// TIA Portal V20 export
VAR_GLOBAL   // PLC tag table "PLC_Production_And_Rework"
   Emergency_Stop_Release AT %I0.0 : Bool;
   Sensor_Water_Fountain_Before_Entrace_Functional_Test_Spinner_Conveyor_Belt AT %I0.1 : Bool;
   Sensor_Water_Fountain_Entrace_Functional_Test_Spinner_Conveyor_Belt AT %I0.2 : Bool;
   Sensor_Water_Fountain_Entrace_Functional_Test_After_Spinner_Conveyor_Belt AT %I0.3 : Bool;
   Trigger_Read_Serial_Number_Entrace_Functional_Test AT %I0.4 : Bool;
   Sensor_Water_Fountain_Geting_Exit_Rework_Conveyor_Belt AT %I0.5 : Bool;
   Button_Water_Fountain_Get_Exit_Rework_Conveyor_Belt AT %I0.6 : Bool;
   Trigger_Read_Serial_Number_Exit_Functional_Test AT %I0.7 : Bool;
   Sensor_Water_Fountain_Exit_Functional_Test_Spinner_Conveyor_Belt AT %I1.0 : Bool;
   Sensor_Water_Fountain_Exit_Functional_Test_After_Spinner_Conveyor_Belt AT %I1.1 : Bool;
   Sensor_Water_Fountain_Geting_Entrace_Rework_Conveyor_Belt_Start AT %I1.2 : Bool;
   Sensor_Water_Fountain_Geting_Entrace_Rework_Conveyor_Belt_Finish AT %I1.3 : Bool;
   Carousel_Frequency_Inverter_Fail AT %I1.4 : Bool;
   Conveyor_Belt_Functional_Test_Inverter_Fail AT %I1.5 : Bool;
   Selected_Voltage_220V AT %I8.0 : Bool;
   Selected_Voltage_127V AT %I8.1 : Bool;
   Sensor_Spinner_Entrace_Functional_Test_Position_Withdrawn AT %I8.2 : Bool;
   Sensor_Spinner_Entrace_Functional_Test_Position_Advanced AT %I8.3 : Bool;
   Sensor_Spinner_Exit_Functional_Test_Position_Withdrawn AT %I8.4 : Bool;
   Sensor_Spinner_Exit_Functional_Test_Position_Advanced AT %I8.5 : Bool;
   Digital_Input_20 AT %I8.6 : Bool;
   Digital_Input_21 AT %I8.7 : Bool;
   Digital_Input_22 AT %I9.0 : Bool;
   Digital_Input_23 AT %I9.1 : Bool;
   Digital_Input_24 AT %I9.2 : Bool;
   Digital_Input_25 AT %I9.3 : Bool;
   Digital_Input_26 AT %I9.4 : Bool;
   Digital_Input_27 AT %I9.5 : Bool;
   Digital_Input_28 AT %I9.6 : Bool;
   Digital_Input_29 AT %I9.7 : Bool;
   Analogic_Input_0 AT %IW64 : Int;
   Analogic_Input_1 AT %IW66 : Int;
   Spin_Carousel_Frequency_Inverter_Speed_1 AT %Q0.0 : Bool;
   Spin_Carousel_Frequency_Inverter_Speed_2 AT %Q0.1 : Bool;
   Spin_Carousel_Frequency_Inverter_Speed_3 AT %Q0.2 : Bool;
   Conveyor_Belt_Frequency_Inverter_Speed_1 AT %Q0.3 : Bool;
   Conveyor_Belt_Frequency_Inverter_Speed_2 AT %Q0.4 : Bool;
   Conveyor_Belt_Frequency_Inverter_Speed_3 AT %Q0.5 : Bool;
   Turn_On_Conveyor_Belt_Motor_Spinner_Get_Entrace_Function_Test AT %Q0.6 : Bool;
   Turn_On_Conveyor_Belt_Motor_Rework_Conveyor_Belt_Get_Entrace_Functional_Test AT %Q0.7 : Bool;
   Turn_On_Conveyor_Belt_Motor_Spinner_Get_Exit_Functional_Test AT %Q1.0 : Bool;
   Turn_On_Conveyor_Belt_Motor_Rework_Conveyor_Belt_Get_Exit_Funcional_Test AT %Q1.1 : Bool;
   Open_Air_Pressure AT %Q8.0 : Bool;
   Valve_Advance_Spinner_Entrace_Functional_Test AT %Q8.1 : Bool;
   Valve_Advance_Spinner_Exit_Functional_Test AT %Q8.2 : Bool;
   Signal_Pre_Functional_Test_Production_Line AT %Q8.3 : Bool;
   Digital_Output_14 AT %Q8.4 : Bool;
   Digital_Output_15 AT %Q8.5 : Bool;
   Digital_Output_16 AT %Q8.6 : Bool;
   Digital_Output_17 AT %Q8.7 : Bool;
   Digital_Output_18 AT %Q9.0 : Bool;
   Digital_Output_19 AT %Q9.1 : Bool;
   Digital_Output_20 AT %Q9.2 : Bool;
   Digital_Output_21 AT %Q9.3 : Bool;
   Digital_Output_22 AT %Q9.4 : Bool;
   Digital_Output_23 AT %Q9.5 : Bool;
   Voltage_220V_Selected AT %Q9.6 : Bool;
   Voltage_127V_Selected AT %Q9.7 : Bool;
   Clock_Byte AT %MB0 : Byte;
   Clock_10Hz AT %M0.0 : Bool;
   Clock_5Hz AT %M0.1 : Bool;
   "Clock_2.5Hz" AT %M0.2 : Bool;
   Clock_2Hz AT %M0.3 : Bool;
   "Clock_1.25Hz" AT %M0.4 : Bool;
   Clock_1Hz AT %M0.5 : Bool;
   "Clock_0.625Hz" AT %M0.6 : Bool;
   "Clock_0.5Hz" AT %M0.7 : Bool;
   System_Byte AT %MB1 : Byte;
   FirstScan AT %M1.0 : Bool;
   DiagStatusUpdate AT %M1.1 : Bool;
   AlwaysTRUE AT %M1.2 : Bool;
   AlwaysFALSE AT %M1.3 : Bool;
END_VAR
